// TIA Portal V20 export
TYPE "typeCmControlNode"
// stored: Namespace Unit1.Em5
   STRUCT
      distanceInPos : Bool;
      interlock : "Unit1.Em5.typeCmControlNodeInterlock";
      command : "Unit1.Em5.typeCmControlNodeCommand";
      softcam : "Unit1.Em5.typeCmControlNodeSoftCam";
      brakeTest : "Unit1.Em5.typeCmControlNodeBrakeTest";
   END_STRUCT;
END_TYPE
